// Mitsubishi GX Works2 project: 7   PLC: FX3U/FX3UC

PROGRAM MAIN
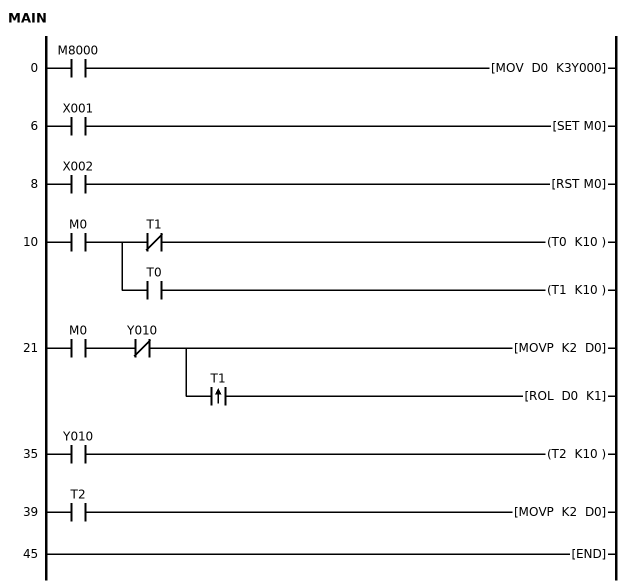
0     LD      M8000
      MOV     D0 K3Y000
6     LD      X001
      SET     M0
8     LD      X002
      RST     M0
10    LD      M0
      MPS
      ANI     T1
      OUT     T0 K10
      MPP
      AND     T0
      OUT     T1 K10
21    LD      M0
      ANI     Y010
      MOVP    K2 D0
      ANDP    T1
      ROL     D0 K1
35    LD      Y010
      OUT     T2 K10
39    LD      T2
      MOVP    K2 D0
45    END
END_PROGRAM
